(*
	Base link component with default interface:
	Control BYTE: From TwinCAT >>> To Unity
	Status BYTE: FROM Unity >>> TO TwinCAT		
*)
FUNCTION_BLOCK FB_LinkDevice EXTENDS FB_Base
VAR		
	{attribute 'simulation_interface'}
	Control		AT %Q* : BYTE;
	{attribute 'simulation_interface'}
	Status		AT %I* : BYTE;
END_VAR

SUPER^();

METHOD INTERNAL GetControl : BYTE
GetControl := Control;
END_METHOD

METHOD INTERNAL SetStatus : BOOL
VAR_INPUT
	nStatus : BYTE;
END_VAR
Status := nStatus;
END_METHOD

END_FUNCTION_BLOCK

(* stored: Version 1.1.0.1, ProductVersion 3.1.4024.12
   POU FB_LinkDevice: Id {898b3300-0d80-065c-002a-6f4eb8497620}, SpecialFunc None
   Method GetControl: Id {4f716504-6ab3-09bf-2b56-18225d9d08da}
   Method SetStatus: Id {8d5d79a5-6c65-0895-3ca9-6c74d83094d8} *)
